# EPICS substitutions: viocs/si_ps/si_psApp/Db/sdp2.substitutions
file "db/individual.db" {
    pattern { family, pos, num }
        { "SDP2", "02C4", "" }
        { "SDP2", "03C1", "" }
        { "SDP2", "06C4", "" }
        { "SDP2", "07C1", "" }
        { "SDP2", "12C4", "" }
        { "SDP2", "11C1", "" }
        { "SDP2", "14C4", "" }
        { "SDP2", "15C1", "" }
        { "SDP2", "18C4", "" }
        { "SDP2", "19C1", "" }
}
